RoboDK station: CAPSTONE_STATION.rdk

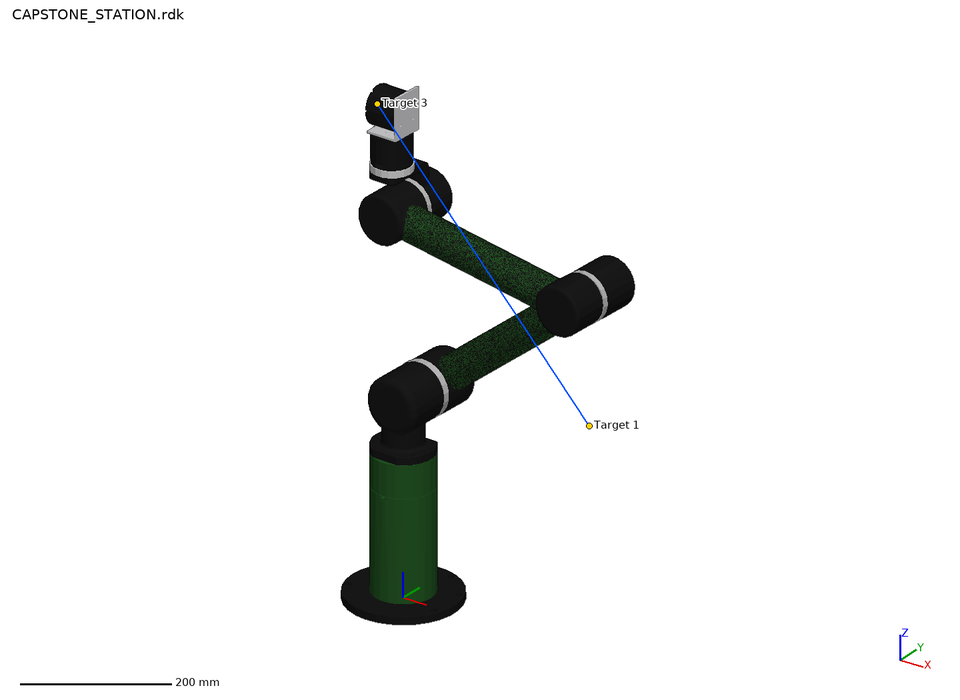
[picture v0: the station drawn from its stored meshes, robots at their saved joint values, targets as dots, program paths as lines]
Station CAPSTONE_STATION (saved by RoboDK 5.9.2). Poses are relative to the parent item; angles as X-Y-Z fixed-axis rotations.
  - frame CAPSTONE_ARM at (0, 0, 0) mm
    - item type 7 CAPSTONE_ARM 基座
    - item type 7 
    - item type 7 
    - item type 7 
    - item type 7 
    - item type 7 
    - item type 7 
  - frame CAPSTONE_ARM 基座 at (0, 0, 0) mm
    - robot CAPSTONE_ARM: 6 axes
        modified DH rows (alpha deg, a mm, theta deg, d mm): 0, 0, 180, 290; 90, 0, 90, 0; 0, 350, 0, 0; 0, 300, -90, 5.65; -90, 0, 180, 154; 90, 0, 0, 23.5
        joint limits [-160, -135, -165, -130, -180, -180] to [160, 135, 165, 130, 180, 180]; home [0, 0, 0, 0, 0, 0]; saved at [-2.726, 51.339, -132.573, 81.034, -89.684, -0.005]
    - target Target 1 (joint target) at (228.02, 101.99, 275.58) mm, rotated rx -90 ry -80 rz 20 deg; joints [-160, -135, 165, -130, 0, 0] of CAPSTONE_ARM
    - target Target 3 (joint target) at (-46.92, 7.76, 708.29) mm, rotated rx 90.2 ry 0 rz -92.41 deg; joints [-2.726, 51.339, -132.573, 81.034, -89.684, -0.005] of CAPSTONE_ARM
  - program 程序1 (3 instructions, listed below)

--- program 程序1 (robot CAPSTONE_ARM) ---
  设置参考: CAPSTONE_ARM 基座
  MoveJ (Target 1)
  MoveJ (Target 3)
